{attribute 'GeneratedUsingTerminal: EL1512-0000-0016'}
{attribute addProperty BoxType "EL1512-0000-0016"}
{attribute addProperty Id "EtcSlaveTerminalBaseCNT_Inputs_Channel_1AT %I*CNT_Inputs_Channel_21E1BB398CNT_Inputs_Channel_2AT %I*CNT_Inputs_Channel_21E1BB398CNT_Outputs_Channel_1AT %Q*CNT_Outputs_Channel_774A30BC6CNT_Outputs_Channel_2AT %Q*CNT_Outputs_Channel_774A30BC6WcStateAT %I*WcState_9091E0EB2InfoDataAT %I*InfoData_32EB74EA10"}
{attribute addProperty CRC "2474461979"}
{attribute addProperty Size "40"}
TYPE EL1512_937D4B1B EXTENDS EtcSlaveTerminalBase :
STRUCT
	{attribute addProperty Name "CNT_Inputs_Channel_1"}
	CNT_Inputs_Channel_1 : CNT_Inputs_Channel_21E1BB39;
	{attribute addProperty Name "CNT_Inputs_Channel_2"}
	CNT_Inputs_Channel_2 : CNT_Inputs_Channel_21E1BB39;
	{attribute addProperty Name "CNT_Outputs_Channel_1"}
	CNT_Outputs_Channel_1 : CNT_Outputs_Channel_774A30BC;
	{attribute addProperty Name "CNT_Outputs_Channel_2"}
	CNT_Outputs_Channel_2 : CNT_Outputs_Channel_774A30BC;
	{attribute addProperty Name "WcState"}
	WcState : WcState_9091E0EB;
	{attribute addProperty Name "InfoData"}
	InfoData : InfoData_32EB74EA;
END_STRUCT
END_TYPE

(* stored: Version 1.2.0.0, ProductVersion 3.1.4024.9
   DUT EL1512_937D4B1B: Id {4e8c551a-c8e5-4332-904e-80a4803c1e66} *)
